// TIA Portal V20 export
DATA_BLOCK "CMInterface_Stirring_DB"   // DB80
// stored: InstanceOfName CM_Interface_Stirring, InstanceOfType FB
"CM_Interface_Stirring"
   // VAR_INPUT
   //    CmCommand { ExternalAccessible := 'False'; ExternalVisible := 'False'; ExternalWritable := 'False'} : Array[0..29] of Bool;
   //    Procedure_Param { ExternalAccessible := 'False'; ExternalVisible := 'False'; ExternalWritable := 'False'} : Array[0..31] of Real;
   //    CmFbOnOff { ExternalAccessible := 'False'; ExternalVisible := 'False'; ExternalWritable := 'False'} : Array[0..29] of Bool;
   //    Pumped_Liters : Real;
   //    Auto_Man : Bool;
   //    Oos : Bool;
   // END_VAR
   // VAR_OUTPUT
   //    CM_E001 { ExternalAccessible := 'False'; ExternalVisible := 'False'; ExternalWritable := 'False'} : "DigVal";
   //    SpeedStirr { ExternalAccessible := 'False'; ExternalVisible := 'False'; ExternalWritable := 'False'} : "AnaVal";
   //    TimeStirr { ExternalAccessible := 'False'; ExternalVisible := 'False'; ExternalWritable := 'False'} : "AnaVal";
   // END_VAR
   // VAR
   //    Neg_edge : Bool;
   //    Pos_edge : Bool;
   // END_VAR
BEGIN
END_DATA_BLOCK
